FUNCTION_BLOCK FB_Test EXTENDS FB_ModeStateControl_Base
VAR_INPUT 
END_VAR
VAR_OUTPUT
END_VAR
VAR
	nCntAuto : UINT;
	nCntManual : UINT;
	nCntMaintenance : UINT;
	
END_VAR


SUPER^.m_Main();

METHOD PUBLIC m_ModeAutomatic : BOOL

nCntAuto := nCntAuto + 1;
END_METHOD

METHOD PUBLIC m_ModeMaintenance : BOOL
VAR_INPUT
END_VAR

nCntMaintenance := nCntMaintenance + 1;
END_METHOD

METHOD PUBLIC m_ModeManual : BOOL
VAR_INPUT
END_VAR

nCntManual := nCntManual + 1;
END_METHOD

END_FUNCTION_BLOCK

(* stored: Version 1.1.0.1, ProductVersion 3.1.4024.12
   POU FB_Test: Id {45bd5caa-5844-4406-ae5b-95c059e1c0cf}, SpecialFunc None
   Method m_ModeAutomatic: Id {df3ea145-7b52-4bc3-8a8d-f96c2a610422}
   Method m_ModeMaintenance: Id {8d071f83-063e-4dd8-b8b9-f394f25423b3}
   Method m_ModeManual: Id {a61bae58-5e3e-4d8b-beaa-08c52286d29b} *)
